// TIA Portal V19 export
TYPE "LAF_typeOperationInterlockInterface"
TITLE = LLGES_OperatorInterlockInterface
// Module interface for external systems
// stored: Access Published
   STRUCT
      commands : "LAF_typeOperationInterlockCommands";
      monitoring { ExternalWritable := 'False'} : "LAF_typeOperationInterlockProcessValues";
   END_STRUCT;
END_TYPE
